TYPE ST_Pressure :
STRUCT
	IN_1St : BOOL;
	IN_2St : BOOL;
	InterlockSt : BOOL;
END_STRUCT
END_TYPE

(* stored: Version 1.1.0.1, ProductVersion 3.1.4024.5
   DUT ST_Pressure: Id {da5f1f5a-107b-4839-97a5-5b6f39fdd832} *)
